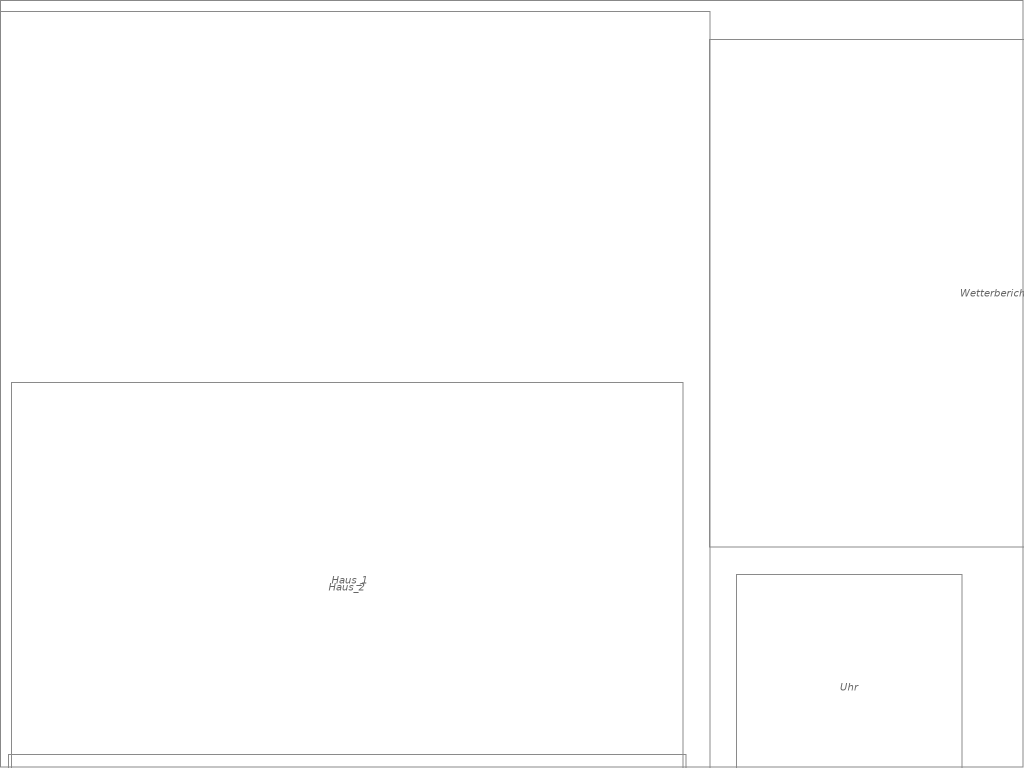
VISUALIZATION MainVisu  // 1024x768
    Frame (-10,11 720x1138), frame switch variable: Simulation
        shows Haus_1()
        shows Simuliertes_Haus()
    Frame (8,754 678x410), invisible if: Simulation
        shows Haus_3()
    Frame (11,382 672x410), invisible if: Simulation
        shows Haus_2()
    Button (1325,51 150x30), "Settings"
        OnMouseClick: OpenDialog Dialog=Settings, OpenModal=True, OpenCentered=True
    Frame (709,39 572x508)
        shows Wetterbericht()
    Frame (713,819 384x276)
        shows Zentrale()
    Button (1327,112 150x30), "Simulation"
        toggle Simulation
        OnMouseClick: OpenDialog Dialog=Simuliertes_Haus, OpenModal=True, PositionX=50, PositionY=50
        OnMouseClick: CloseDialog Dialog=Simuliertes_Haus, Result=OK, NumpadKeypadSet=True
    Frame (736,574 226x226)
        shows Uhr()
END_VISUALIZATION

(* stored: Version 1.1.0.1, ProductVersion 3.1.4018.5
   Visu MainVisu: Id {1793421b-1095-4da5-bbbd-8fc376f66a69} *)
